% RSLogix 500 project ELEVATOR.RSS, saved by version 8.30.00.16 %
PROJECT "UNTITLED"    % processor: Bul.1763 MicroLogix 1100 Series B %

PROGRAM FILES
  LAD 2   19 rungs

DATA FILES
  O0 OUTPUT  4 elements
  I1 INPUT  6 elements
  S2 STATUS  66 elements
  B3 BINARY  2 elements
  T4 TIMER  1 elements
  C5 COUNTER  1 elements
  R6 CONTROL  1 elements
  N7 INTEGER  1 elements
  F8 FLOAT  1 elements

LADDER 2
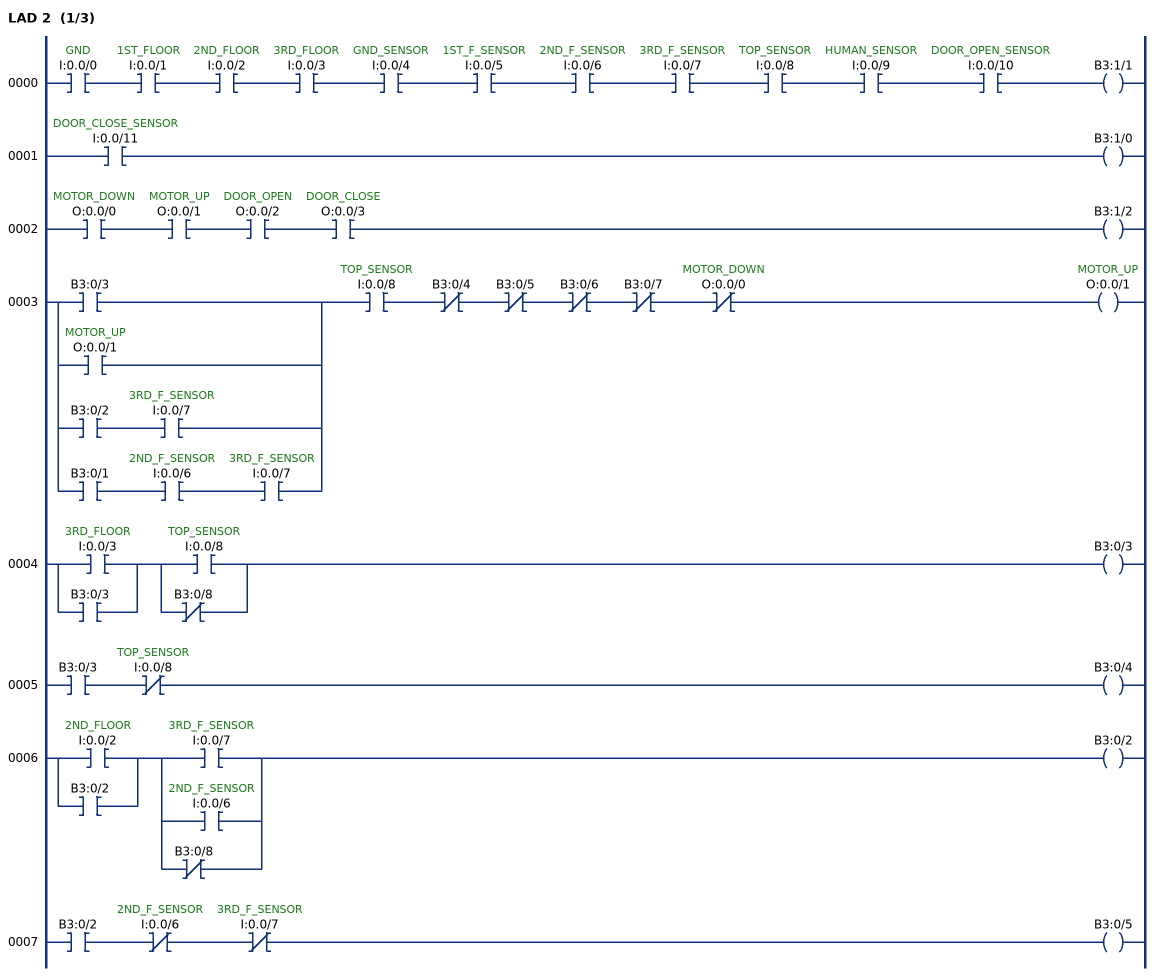
% Rung: 0 %
SOR XIC I:0.0/0 XIC I:0.0/1 XIC I:0.0/2 XIC I:0.0/3 XIC I:0.0/4 XIC I:0.0/5 XIC I:0.0/6 XIC I:0.0/7 XIC I:0.0/8 XIC I:0.0/9 XIC I:0.0/10 OTE B3:1/1 EOR
%   I:0.0/0  GND %
%   I:0.0/1  1ST_FLOOR %
%   I:0.0/2  2ND_FLOOR %
%   I:0.0/3  3RD_FLOOR %
%   I:0.0/4  GND_SENSOR %
%   I:0.0/5  1ST_F_SENSOR %
%   I:0.0/6  2ND_F_SENSOR %
%   I:0.0/7  3RD_F_SENSOR %
%   I:0.0/8  TOP_SENSOR %
%   I:0.0/9  HUMAN_SENSOR %
%   I:0.0/10  DOOR_OPEN_SENSOR %
% Rung: 1 %
SOR XIC I:0.0/11 OTE B3:1/0 EOR
%   I:0.0/11  DOOR_CLOSE_SENSOR %
% Rung: 2 %
SOR XIC O:0.0/0 XIC O:0.0/1 XIC O:0.0/2 XIC O:0.0/3 OTE B3:1/2 EOR
%   O:0.0/0  MOTOR_DOWN %
%   O:0.0/1  MOTOR_UP %
%   O:0.0/2  DOOR_OPEN %
%   O:0.0/3  DOOR_CLOSE %
% Rung: 3 %
SOR BST BST XIC B3:0/3 NXB XIC O:0.0/1 BND NXB BST XIC B3:0/2 XIC I:0.0/7 NXB XIC B3:0/1 XIC I:0.0/6 XIC I:0.0/7 BND BND XIC I:0.0/8 XIO B3:0/4 XIO B3:0/5 XIO B3:0/6 XIO B3:0/7 XIO O:0.0/0 OTE O:0.0/1 EOR
%   O:0.0/1  MOTOR_UP %
%   I:0.0/7  3RD_F_SENSOR %
%   I:0.0/6  2ND_F_SENSOR %
%   I:0.0/8  TOP_SENSOR %
%   O:0.0/0  MOTOR_DOWN %
% Rung: 4 %
SOR BST XIC I:0.0/3 NXB XIC B3:0/3 BND BST XIC I:0.0/8 NXB XIO B3:0/8 BND OTE B3:0/3 EOR
%   I:0.0/3  3RD_FLOOR %
%   I:0.0/8  TOP_SENSOR %
% Rung: 5 %
SOR XIC B3:0/3 XIO I:0.0/8 OTE B3:0/4 EOR
%   I:0.0/8  TOP_SENSOR %
% Rung: 6 %
SOR BST XIC I:0.0/2 NXB XIC B3:0/2 BND BST XIC I:0.0/7 NXB BST XIC I:0.0/6 NXB XIO B3:0/8 BND BND OTE B3:0/2 EOR
%   I:0.0/2  2ND_FLOOR %
%   I:0.0/7  3RD_F_SENSOR %
%   I:0.0/6  2ND_F_SENSOR %
% Rung: 7 %
SOR XIC B3:0/2 XIO I:0.0/6 XIO I:0.0/7 OTE B3:0/5 EOR
%   I:0.0/6  2ND_F_SENSOR %
%   I:0.0/7  3RD_F_SENSOR %

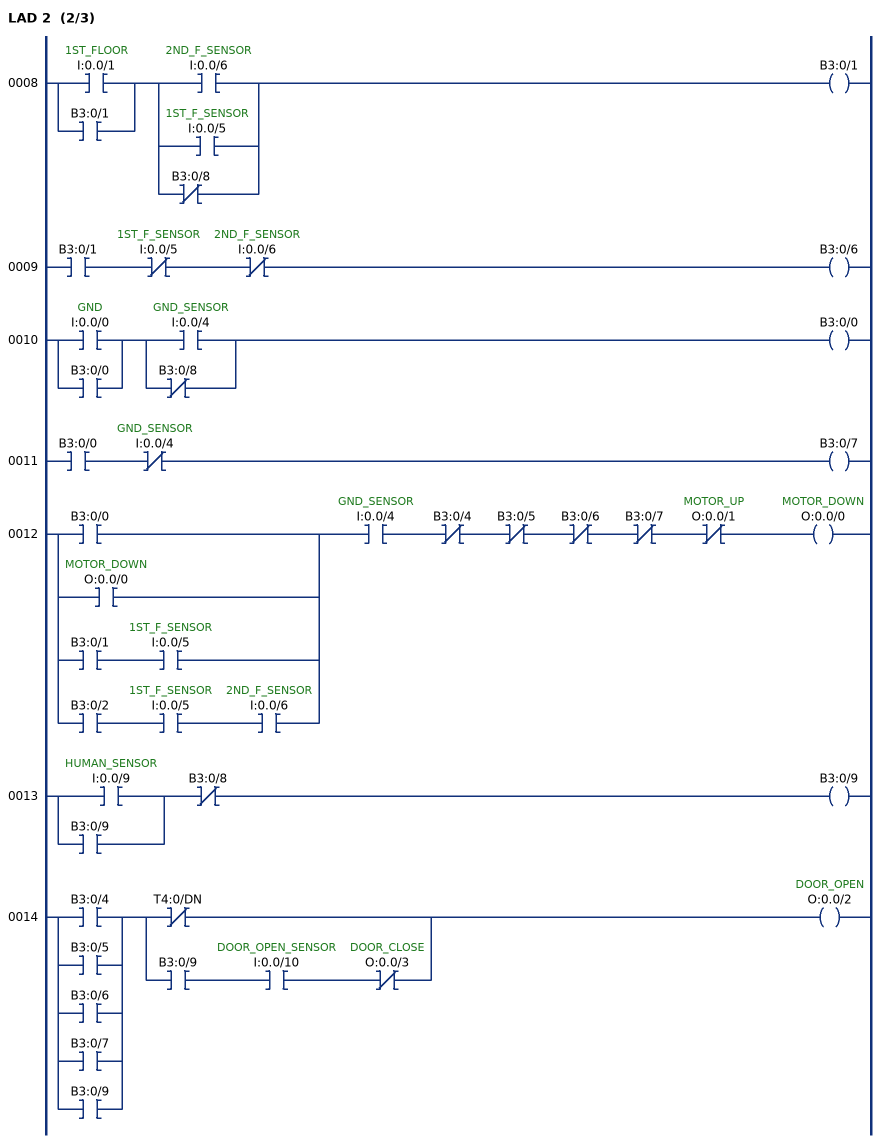
% Rung: 8 %
SOR BST XIC I:0.0/1 NXB XIC B3:0/1 BND BST XIC I:0.0/6 NXB BST XIC I:0.0/5 NXB XIO B3:0/8 BND BND OTE B3:0/1 EOR
%   I:0.0/1  1ST_FLOOR %
%   I:0.0/6  2ND_F_SENSOR %
%   I:0.0/5  1ST_F_SENSOR %
% Rung: 9 %
SOR XIC B3:0/1 XIO I:0.0/5 XIO I:0.0/6 OTE B3:0/6 EOR
%   I:0.0/5  1ST_F_SENSOR %
%   I:0.0/6  2ND_F_SENSOR %
% Rung: 10 %
SOR BST XIC I:0.0/0 NXB XIC B3:0/0 BND BST XIC I:0.0/4 NXB XIO B3:0/8 BND OTE B3:0/0 EOR
%   I:0.0/0  GND %
%   I:0.0/4  GND_SENSOR %
% Rung: 11 %
SOR XIC B3:0/0 XIO I:0.0/4 OTE B3:0/7 EOR
%   I:0.0/4  GND_SENSOR %
% Rung: 12 %
SOR BST BST XIC B3:0/0 NXB XIC O:0.0/0 BND NXB BST XIC B3:0/1 XIC I:0.0/5 NXB XIC B3:0/2 XIC I:0.0/5 XIC I:0.0/6 BND BND XIC I:0.0/4 XIO B3:0/4 XIO B3:0/5 XIO B3:0/6 XIO B3:0/7 XIO O:0.0/1 OTE O:0.0/0 EOR
%   O:0.0/0  MOTOR_DOWN %
%   I:0.0/5  1ST_F_SENSOR %
%   I:0.0/6  2ND_F_SENSOR %
%   I:0.0/4  GND_SENSOR %
%   O:0.0/1  MOTOR_UP %
% Rung: 13 %
SOR BST XIC I:0.0/9 NXB XIC B3:0/9 BND XIO B3:0/8 OTE B3:0/9 EOR
%   I:0.0/9  HUMAN_SENSOR %
% Rung: 14 %
SOR BST XIC B3:0/4 NXB BST XIC B3:0/5 NXB BST XIC B3:0/6 NXB BST XIC B3:0/7 NXB XIC B3:0/9 BND BND BND BND BST XIO T4:0/DN NXB XIC B3:0/9 XIC I:0.0/10 XIO O:0.0/3 BND OTE O:0.0/2 EOR
%   I:0.0/10  DOOR_OPEN_SENSOR %
%   O:0.0/3  DOOR_CLOSE %
%   O:0.0/2  DOOR_OPEN %

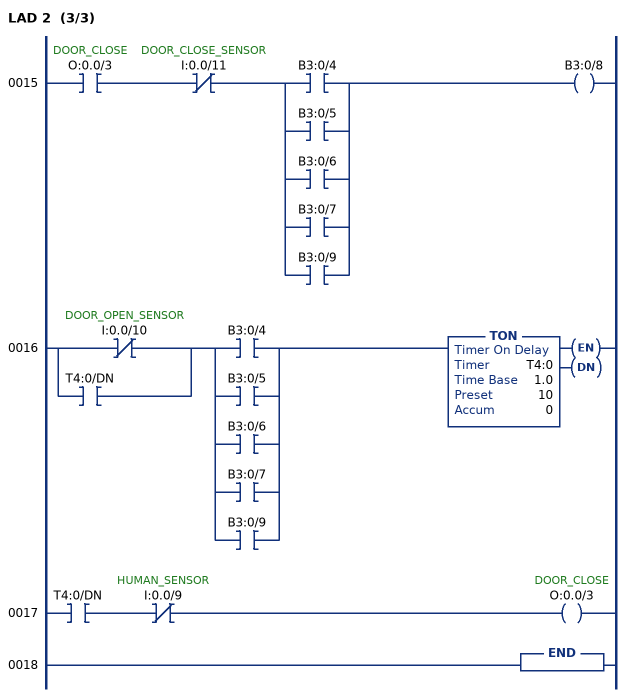
% Rung: 15 %
SOR XIC O:0.0/3 XIO I:0.0/11 BST XIC B3:0/4 NXB BST XIC B3:0/5 NXB BST XIC B3:0/6 NXB BST XIC B3:0/7 NXB XIC B3:0/9 BND BND BND BND OTE B3:0/8 EOR
%   O:0.0/3  DOOR_CLOSE %
%   I:0.0/11  DOOR_CLOSE_SENSOR %
% Rung: 16 %
SOR BST XIO I:0.0/10 NXB XIC T4:0/DN BND BST XIC B3:0/4 NXB BST XIC B3:0/5 NXB BST XIC B3:0/6 NXB BST XIC B3:0/7 NXB XIC B3:0/9 BND BND BND BND TON T4:0 1.0 10 0 EOR
%   I:0.0/10  DOOR_OPEN_SENSOR %
% Rung: 17 %
SOR XIC T4:0/DN XIO I:0.0/9 OTE O:0.0/3 EOR
%   I:0.0/9  HUMAN_SENSOR %
%   O:0.0/3  DOOR_CLOSE %
% Rung: 18 %
SOR END EOR

OTHER DOCUMENTED ADDRESSES
  C0  

DATA TABLE (non-zero values as saved)
DATA B3
% B3:0 % 0X0001 0X0000
DATA T4
% .PRE .ACC %
% T4:0 % 10 0
DATA C5
% .PRE .ACC %
% C5:0 % 10 8
